(* CODESYS project 2021_06_14_Gr2_SPS_Göller_Huang_Troll.project

Project tree, tasks and I/O mapping:
  Device : CODESYS Control Win V3, 3S - Smart Software Solutions GmbH, order no. 305021, version 3.5.10.20
    application Application
      libraries: Standard, * (System)
      task Task (freewheeling, priority 1) calls PLG_PROG
      task VISU_TASK (cyclic, interval 100 ms, priority 31) calls VisuElems.Visu_Prg
      visualisation Visualization
  libraries: AC_ModuleBase, * (3S - Smart Software Solutions GmbH); AC_DeviceDiagnosis, 3.5.9.0 (3S - Smart Software Solutions GmbH); AC_Persistence, 3.5.10.0 (3S - Smart Software Solutions GmbH); VisuSymbols, 3.5.10.0 (System)
  global variables GVL
  program PLG_PROG [CFC]
  program TrafficLight_Cars [FBD]
  program TrafficLight_Control [SFC]: KFZ_rotgelb_FG_rot_active, T1s, KFZ_gruen_FG_rot_active, KFZ_rot_FG_rot_active, T3s, KFZ_gelb_FG_rot_active, Init_active, KFZ_rot_FG_gruen_active, KFZ_rot_FG_rot_2_active, T5s, T2s, T4s, off, Auszustand_active_0, signal, gelb_an_active, gelb_aus_active
  program Eingang [FBD]
  program TrafficLight_FG [FBD]
  text list GlobalTextList
*)

// GVL
{attribute 'qualified_only'}
VAR_GLOBAL
	
	on:BOOL:=0;
	ereig:BOOL:=0;
	nacht:BOOL:=0;
	
	rot_KFZ: BOOL;
	gelb_KFZ: BOOL;
	gruen_KFZ: BOOL;
	rot_FG: BOOL;
	gruen_FG: BOOL;
END_VAR

// PLG_PROG
PROGRAM PLG_PROG

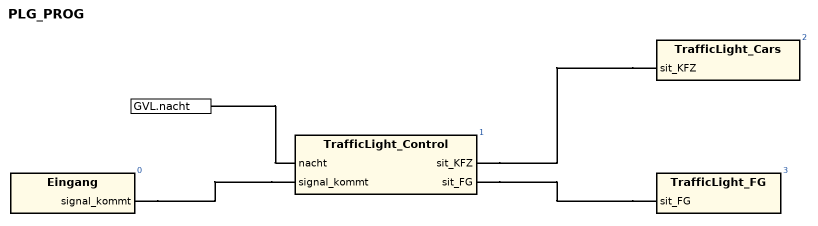
Eingang();
TrafficLight_Control(nacht := GVL.nacht, signal_kommt := Eingang.signal_kommt);
TrafficLight_Cars(sit_KFZ := TrafficLight_Control.sit_KFZ);
TrafficLight_FG(sit_FG := TrafficLight_Control.sit_FG);

END_PROGRAM

// Eingang
PROGRAM Eingang
VAR
	RS_ereignis:RS;
END_VAR
VAR_OUTPUT
	signal_kommt:BOOL;
	
END_VAR

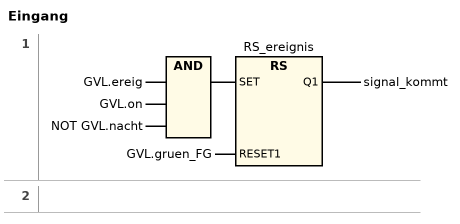
// NETWORK 1
RS_ereignis(SET := GVL.ereig AND GVL.on AND (NOT GVL.nacht), RESET1 := GVL.gruen_FG); // RS
signal_kommt := RS_ereignis.Q1;

// NETWORK 2

END_PROGRAM

// TrafficLight_Control
PROGRAM TrafficLight_Control
VAR_OUTPUT
	sit_KFZ: INT;
	sit_FG: INT;
END_VAR

VAR_INPUT
	nacht:BOOL;
	signal_kommt:BOOL;
END_VAR

VAR
	delay1: BOOL;
	delay_gelb: BOOL;
	delay_gelb_aus: BOOL;
END_VAR

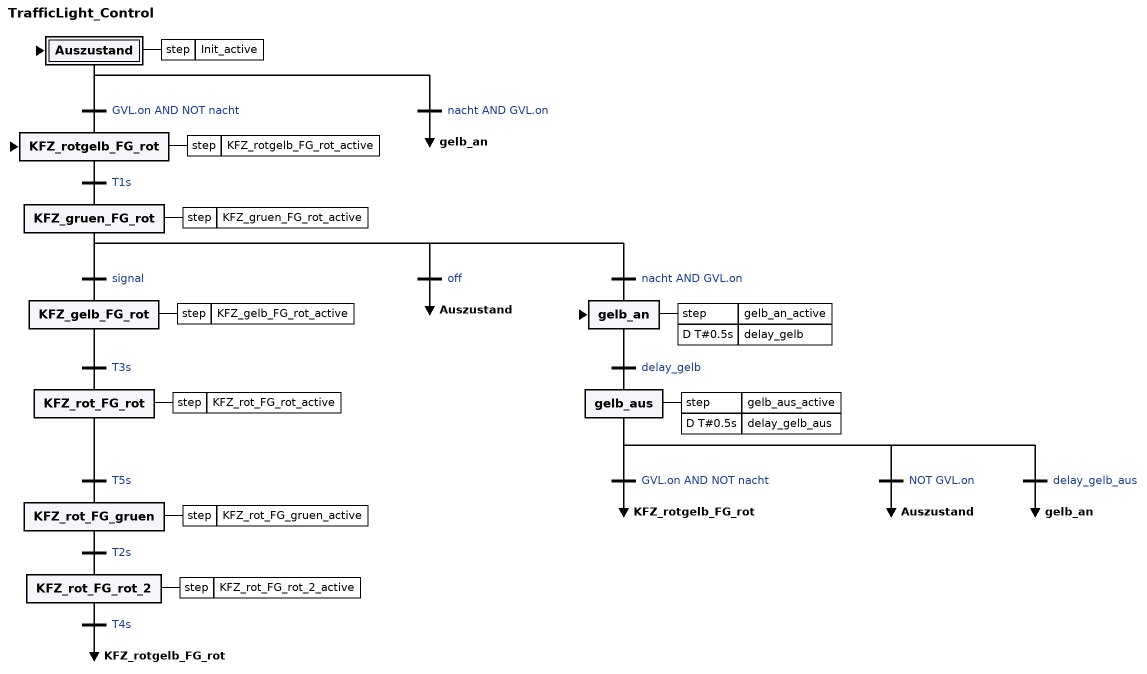
INITIAL_STEP Auszustand:
    Init_active(N);  // step action
END_STEP
TRANSITION FROM Auszustand TO KFZ_rotgelb_FG_rot
    := GVL.on AND NOT nacht;
END_TRANSITION
TRANSITION FROM Auszustand TO gelb_an
    := nacht AND GVL.on;
END_TRANSITION
STEP KFZ_rotgelb_FG_rot:
    KFZ_rotgelb_FG_rot_active(N);  // step action
END_STEP
TRANSITION FROM KFZ_rotgelb_FG_rot TO KFZ_gruen_FG_rot
    := T1s;
END_TRANSITION
STEP KFZ_gruen_FG_rot:
    KFZ_gruen_FG_rot_active(N);  // step action
END_STEP
TRANSITION FROM KFZ_gruen_FG_rot TO KFZ_gelb_FG_rot
    := signal;
END_TRANSITION
TRANSITION FROM KFZ_gruen_FG_rot TO Auszustand
    := off;
END_TRANSITION
TRANSITION FROM KFZ_gruen_FG_rot TO gelb_an
    := nacht AND GVL.on;
END_TRANSITION
STEP gelb_an:
    gelb_an_active(N);  // step action
    delay_gelb(D, T#0.5s);
END_STEP
TRANSITION FROM gelb_an TO gelb_aus
    := delay_gelb;
END_TRANSITION
STEP gelb_aus:
    gelb_aus_active(N);  // step action
    delay_gelb_aus(D, T#0.5s);
END_STEP
TRANSITION FROM gelb_aus TO KFZ_rotgelb_FG_rot
    := GVL.on AND NOT nacht;
END_TRANSITION
TRANSITION FROM gelb_aus TO Auszustand
    := NOT GVL.on;
END_TRANSITION
TRANSITION FROM gelb_aus TO gelb_an
    := delay_gelb_aus;
END_TRANSITION
STEP KFZ_gelb_FG_rot:
    KFZ_gelb_FG_rot_active(N);  // step action
END_STEP
TRANSITION FROM KFZ_gelb_FG_rot TO KFZ_rot_FG_rot
    := T3s;
END_TRANSITION
STEP KFZ_rot_FG_rot:
    KFZ_rot_FG_rot_active(N);  // step action
END_STEP
TRANSITION FROM KFZ_rot_FG_rot TO KFZ_rot_FG_gruen
    := T5s;
END_TRANSITION
STEP KFZ_rot_FG_gruen:
    KFZ_rot_FG_gruen_active(N);  // step action
END_STEP
TRANSITION FROM KFZ_rot_FG_gruen TO KFZ_rot_FG_rot_2
    := T2s;
END_TRANSITION
STEP KFZ_rot_FG_rot_2:
    KFZ_rot_FG_rot_2_active(N);  // step action
END_STEP
TRANSITION FROM KFZ_rot_FG_rot_2 TO KFZ_rotgelb_FG_rot
    := T4s;
END_TRANSITION

ACTION KFZ_rotgelb_FG_rot_active:
sit_KFZ:=0;
sit_FG:=0;
END_ACTION

TRANSITION T1s:
KFZ_rotgelb_FG_rot.t > T#1S;
END_TRANSITION

ACTION KFZ_gruen_FG_rot_active:
sit_KFZ:=1;
sit_FG:=0;
END_ACTION

ACTION KFZ_rot_FG_rot_active:
sit_KFZ:=3;
sit_FG:=0;
END_ACTION

TRANSITION T3s:
KFZ_gelb_FG_rot.t >=T#3s;
END_TRANSITION

ACTION KFZ_gelb_FG_rot_active:
sit_KFZ:=2;
sit_FG:=0;
END_ACTION

ACTION Init_active:
sit_KFZ:=4;
sit_FG:=2;
signal_kommt:=FALSE;
END_ACTION

ACTION KFZ_rot_FG_gruen_active:
sit_KFZ:=3;
sit_FG:=1;
END_ACTION

ACTION KFZ_rot_FG_rot_2_active:
sit_KFZ:=3;
sit_FG:=0;
END_ACTION

TRANSITION T5s:
KFZ_rot_FG_rot.t> T#5S;
END_TRANSITION

TRANSITION T2s:
KFZ_rot_FG_gruen.t> T#2s;
END_TRANSITION

TRANSITION T4s:
(KFZ_rot_FG_rot_2.t > T#4s);
END_TRANSITION

TRANSITION off:
GVL.on=FALSE AND KFZ_gruen_FG_rot.t >=T#1S;
END_TRANSITION

ACTION Auszustand_active_0:
sit_KFZ:=4;
sit_FG:=2;
END_ACTION

TRANSITION signal:
KFZ_gruen_FG_rot.t >=T#5s AND signal_kommt;
END_TRANSITION

ACTION gelb_an_active:
sit_KFZ:=2;
sit_FG:=2;
END_ACTION

ACTION gelb_aus_active:
sit_KFZ:=4;
sit_FG:=2;
END_ACTION

END_PROGRAM

// TrafficLight_Cars
PROGRAM TrafficLight_Cars


VAR_INPUT
	sit_KFZ:INT;
END_VAR

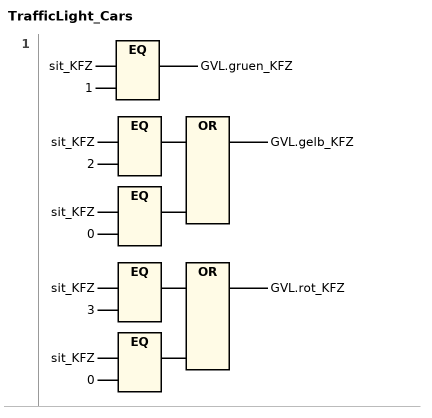
// NETWORK 1
GVL.gruen_KFZ := sit_KFZ = 1;
GVL.gelb_KFZ := sit_KFZ = 2 OR sit_KFZ = 0;
GVL.rot_KFZ := sit_KFZ = 3 OR sit_KFZ = 0;

END_PROGRAM

// TrafficLight_FG
PROGRAM TrafficLight_FG

VAR_INPUT
	sit_FG:INT;
END_VAR

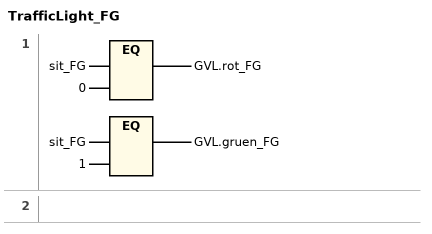
// NETWORK 1
GVL.rot_FG := sit_FG = 0;
GVL.gruen_FG := sit_FG = 1;

// NETWORK 2

END_PROGRAM

// Device/Application/Visualization
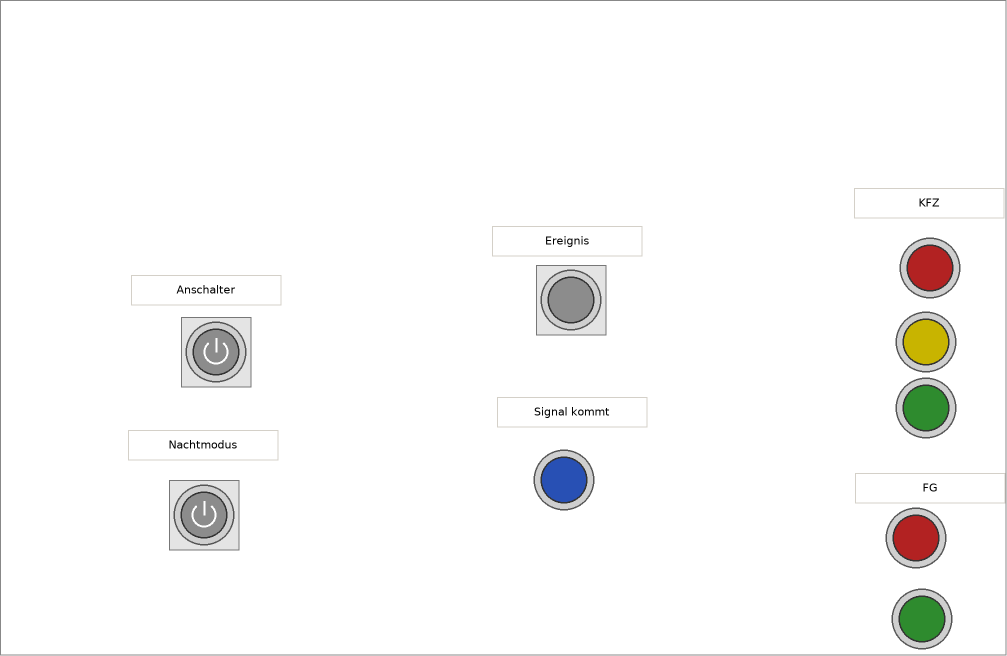
VISUALIZATION Visualization  // 1007x656
    PushSwitch (536,265 70x70), tooltip "Ereignis", variable: GVL.ereig, behaviour: TAP, style: Switch-PushSwitch-Gray
    PowerSwitch (181,317 70x70), variable: GVL.on, behaviour: TOGGLE, style: Switch-PowerSwitch-Gray
    Lamp1 (895,233 70x70), variable: GVL.rot_KFZ, style: Lamp-Lamp1-Red
    Lamp1 (891,307 70x70), variable: GVL.gelb_KFZ, style: Lamp-Lamp1-Yellow
    Lamp1 (891,373 70x70), variable: GVL.gruen_KFZ, style: Lamp-Lamp1-Green
    Lamp1 (881,503 70x70), variable: GVL.rot_FG, style: Lamp-Lamp1-Red
    Lamp1 (887,584 70x70), variable: GVL.gruen_FG, style: Lamp-Lamp1-Green
    Textfield (131,275 150x30), "Anschalter"
    Textfield (492,226 150x30), "Ereignis"
    Textfield (854,188 150x30), "KFZ"
    Textfield (855,473 150x30), "FG"
    Lamp1 (529,445 70x70), variable: TrafficLight_Control.signal_kommt, style: Lamp-Lamp1-Blue
    Textfield (497,397 150x30), "Signal kommt"
    PowerSwitch (169,480 70x70), variable: GVL.nacht, behaviour: TOGGLE, style: Switch-PowerSwitch-Gray
    Textfield (128,430 150x30), "Nachtmodus"
END_VISUALIZATION
